(* CODESYS project 1002_xlh_stamp_button_switch_led_manager.project
   Description: Receives some incoming messages and echoes them with CAN-ID +1
   Company: 3S - Smart Software Solutions GmbH
   Version: 1.0.0.0
   Title: CAN Bus API Example
   Author: 3S - Smart Software Solutions GmbH

Project tree, tasks and I/O mapping:
  xLH_base : CODESYS Control for Raspberry Pi 64 SL, CODESYS, order no. 2302000009, version 4.18.0.0
    application app
      libraries: Standard, 3.5.18.0 (System); Util, 3.5.21.0 (System); VisuDialogs, * (System); Memory, * (3S - Smart Software Solutions GmbH); CmpBitmapPool, * (System); CAN API, 1.0.0.4 (CODESYS); MemoryUtils, * (3S - Smart Software Solutions GmbH); CAA CiA 405, 4.3.0.0 (CODESYS)
      task MAIN_TASK (cyclic, interval 10 ms, priority 1) calls ExpeditedReadExample, MAIN
      program MAIN [ST]
      trace Trace_Switch (task MAIN_TASK): MAIN.byDigOutButton, MAIN.byDigInButton, MAIN.fbReadStatusLoopTime.diValue
      function block FB_SDO_READ_4_BYTE [ST]
      CO_API/
        program ExpeditedReadExample [ST]
        program ExpeditedWriteExample [ST]
    SoftMotion General Axis Pool
      a_axis : SM_Drive_PosControl, CODESYS, order no. 1805, version 4.18.0.0
          settings: wDriveID = 4; dwRatioTechUnitsDenom = 101846; iRatioTechUnitsNum = -125; eRampType = 1; fSWMaxVelocity = 50; fSWMaxAcceleration = 100; fSWMaxDeceleration = 100; fSWMaxJerk = 1000; fSWLimitNegative = -1000.0; ScalingIncs = 814768; ScalingUnits = 1000; InvertDirection = TRUE; IsLinearMotor = TRUE; MaximumOutputVelocityInt = 40738; MinimumOutputVelocityInt = -40738; Kp = 0.05; MaxFollowingError = 5.0; EnableFollowingErrorCheck = TRUE; DeadTime = 3.0
      x_axis : SM_Drive_PosControl, CODESYS, order no. 1805, version 4.18.0.0
          settings: dwRatioTechUnitsDenom = 101846; iRatioTechUnitsNum = 125; eRampType = 1; fSWMaxVelocity = 50; fSWMaxAcceleration = 100; fSWMaxDeceleration = 100; fSWMaxJerk = 1000; fSWLimitNegative = -1000; ScalingIncs = 814768; ScalingUnits = 1000; IsLinearMotor = TRUE; MaximumOutputVelocityInt = 40738; MinimumOutputVelocityInt = -40738; Kp = 0.05; MaxFollowingError = 5.0; EnableFollowingErrorCheck = TRUE; DeadTime = 3.0
      y_axis : SM_Drive_PosControl, CODESYS, order no. 1805, version 4.18.0.0
          settings: wDriveID = 2; dwRatioTechUnitsDenom = 101846; iRatioTechUnitsNum = 125; eRampType = 1; fSWMaxVelocity = 50; fSWMaxAcceleration = 100; fSWMaxDeceleration = 100; fSWMaxJerk = 1000; fSWLimitNegative = -1000; ScalingIncs = 814768; ScalingUnits = 1000; IsLinearMotor = TRUE; MaximumOutputVelocityInt = 40738; MinimumOutputVelocityInt = -40738; Kp = 0.05; MaxFollowingError = 5.0; EnableFollowingErrorCheck = TRUE; DeadTime = 3.0
      z_axis : SM_Drive_PosControl, CODESYS, order no. 1805, version 4.18.0.0
          settings: wDriveID = 3; dwRatioTechUnitsDenom = 101846; iRatioTechUnitsNum = 125; eRampType = 1; fSWMaxVelocity = 50; fSWMaxAcceleration = 100; fSWMaxDeceleration = 100; fSWMaxJerk = 1000; fSWLimitNegative = -1000; ScalingIncs = 814768; ScalingUnits = 1000; IsLinearMotor = TRUE; MaximumOutputVelocityInt = 40738; MinimumOutputVelocityInt = -40738; Kp = 0.05; MaxFollowingError = 5.0; EnableFollowingErrorCheck = TRUE; DeadTime = 3.0
    GPIOs_A_B : GPIOs B+/Pi2, CODESYS, version 4.18.0.0
        unmapped channels: digital inputs (GPIO0..GPIO31), digital outputs (GPIO0..GPIO31)
    Onewire
    Camera device
      <Leer>
    SPI
    I²C
    CANbus : CANbus, CODESYS, version 4.3.0.0
        settings: Baudrate = 1000 kbit/s
      CANopen_Manager : CANopen_Manager, CODESYS, version 4.3.0.0
          settings: ConfigVersion = 50659584
        xlh_digital_switch_button_led : xlh_digital_switch_button_led, xemax ag, order no. 0, version Revision=16#00000001, FileVersion=1.0
            settings: NODEIDSAVED = 1; SDO Timeout = 1000000; PDO_Autoconfig = FALSE; EXPERTSETTINGS = False; Sync-General Parameters.Sync-COBID = 16#00000080; Sync-General Parameters.Communication Cycle Period = 16#00000000 usec; PDO 16#1400.COBID = 16#00000201; Process by CANopenManager = TRUE; PDO 16#1800.COBID = 16#00000181; Process by CANopenManager = TRUE; Leds Button.Subindex = 16#01; Leds Switch.Subindex = 16#01; Digital Inputs Button.Subindex = 16#01; Digital Inputs Switch.Subindex = 16#01; SDO List.Set COB-ID sync.Index = 16#1005; SDO List.Set COB-ID sync.Subindex = 16#00; SDO List.Set COB-ID sync.Value = 16#00000080; SDO List.Set COB-ID sync.Size = 32; SDO List.Set COB-ID sync.AbortIfError = FALSE; SDO List.Set COB-ID sync.JumpToLine = FALSE; SDO List.Set COB-ID sync.Line = 0; SDO List.Set communication cycle period.Index = 16#1006; SDO List.Set communication cycle period.Subindex = 16#00; SDO List.Set communication cycle period.Value = 16#00000000; SDO List.Set communication cycle period.Size = 32; SDO List.Set communication cycle period.AbortIfError = FALSE; SDO List.Set communication cycle period.JumpToLine = FALSE; SDO List.Set communication cycle period.Line = 0; SDO List.Set Guardtime.Index = 16#100C; SDO List.Set Guardtime.Subindex = 16#00; SDO List.Set Guardtime.Value = 16#000000C8; SDO List.Set Guardtime.Size = 16; SDO List.Set Guardtime.AbortIfError = FALSE; SDO List.Set Guardtime.JumpToLine = FALSE; SDO List.Set Guardtime.Line = 0; SDO List.Set Lifetime.Index = 16#100D; SDO List.Set Lifetime.Subindex = 16#00; SDO List.Set Lifetime.Value = 16#00000003; SDO List.Set Lifetime.Size = 8; SDO List.Set Lifetime.AbortIfError = FALSE;
              SDO List.Set Lifetime.JumpToLine = FALSE; SDO List.Set Lifetime.Line = 0; SDO List.Set Heartbeat Consumer.Index = 16#1016; SDO List.Set Heartbeat Consumer.Subindex = 16#01; SDO List.Set Heartbeat Consumer.Value = 0; SDO List.Set Heartbeat Consumer.Size = 32; SDO List.Set Heartbeat Consumer.AbortIfError = FALSE; SDO List.Set Heartbeat Consumer.JumpToLine = FALSE; SDO List.Set Heartbeat Consumer.Line = 0; SDO List.Disable PDO.Index = 16#1400; SDO List.Disable PDO.Subindex = 16#01; SDO List.Disable PDO.Value = 16#80000201; SDO List.Disable PDO.Size = 32; SDO List.Disable PDO.AbortIfError = FALSE; SDO List.Disable PDO.JumpToLine = FALSE; SDO List.Disable PDO.Line = 0; SDO List.Set transmission type.Index = 16#1400; SDO List.Set transmission type.Subindex = 16#02; SDO List.Set transmission type.Value = 16#FF; SDO List.Set transmission type.Size = 8; SDO List.Set transmission type.AbortIfError = FALSE; SDO List.Set transmission type.JumpToLine = FALSE; SDO List.Set transmission type.Line = 0; SDO List.Set and enable COB-ID.Index = 16#1400; SDO List.Set and enable COB-ID.Subindex = 16#01; SDO List.Set and enable COB-ID.Value = 16#00000201; SDO List.Set and enable COB-ID.Size = 32; SDO List.Set and enable COB-ID.AbortIfError = FALSE; SDO List.Set and enable COB-ID.JumpToLine = FALSE; SDO List.Set and enable COB-ID.Line = 0; SDO List.Disable PDO.Index = 16#1800; SDO List.Disable PDO.Subindex = 16#01; SDO List.Disable PDO.Value = 16#80000181; SDO List.Disable PDO.Size = 32; SDO List.Disable PDO.AbortIfError = FALSE; SDO List.Disable PDO.JumpToLine = FALSE; SDO List.Disable PDO.Line = 0; SDO List.Set transmission type.Index = 16#1800; SDO List.Set transmission type.Subindex = 16#02; SDO List.Set transmission type.Value = 16#FF;
              SDO List.Set transmission type.Size = 8; SDO List.Set transmission type.AbortIfError = FALSE; SDO List.Set transmission type.JumpToLine = FALSE; SDO List.Set transmission type.Line = 0; SDO List.Set inhibit time.Index = 16#1800; SDO List.Set inhibit time.Subindex = 16#03; SDO List.Set inhibit time.Value = 16#0000; SDO List.Set inhibit time.Size = 16; SDO List.Set inhibit time.AbortIfError = FALSE; SDO List.Set inhibit time.JumpToLine = FALSE; SDO List.Set inhibit time.Line = 0; SDO List.Set event time.Index = 16#1800; SDO List.Set event time.Subindex = 16#05; SDO List.Set event time.Value = 16#0000; SDO List.Set event time.Size = 16; SDO List.Set event time.AbortIfError = FALSE; SDO List.Set event time.JumpToLine = FALSE; SDO List.Set event time.Line = 0; SDO List.Set and enable COB-ID.Index = 16#1800; SDO List.Set and enable COB-ID.Subindex = 16#01; SDO List.Set and enable COB-ID.Value = 16#00000181; SDO List.Set and enable COB-ID.Size = 32; SDO List.Set and enable COB-ID.AbortIfError = FALSE; SDO List.Set and enable COB-ID.JumpToLine = FALSE; SDO List.Set and enable COB-ID.Line = 0; ConfigVersion = 50659584
            output app.MAIN.byDigOutButton : USINT  // Digital Outputs Button
            output app.MAIN.byDigOutSwitch : USINT  // Digital Outputs Switch
            input  app.MAIN.byDigInButton : USINT  // Digital Inputs Button
            input  app.MAIN.byDigInSwitch : USINT  // Digital Inputs Switch
  libraries: VisuSymbols, 4.5.0.0 (System); DepictorBase, 1.2.0.0 (CODESYS)
  text list GlobalTextList
  5ce3da45-db07-42e7-a21c-a00fff4ed8f6|C:\Users\phe\Downloads\Musterloesung_FUP.PNG
*)

// xLH_base/app/CO_API/ExpeditedReadExample
// The following program reads the device type of CANopenRemoteDevice and shows how to usde SDORead4 function block.
// Set xEnable to TRUE in online mode to get the program working.
PROGRAM ExpeditedReadExample
VAR
	xEnable       : BOOL; // Set this variable to true to start the example code. Variable will be set to FALSE if Expedited transfer finished execution.
	dwValue : DWORD; //read value
	dwAbortCode : DWORD; //contains abort code in case of error
	
	SDORead4 	  : CIA405.SDO_READ4;
END_VAR

IF SDORead4.CONFIRM THEN
	//value was read without error
	// ==> Copy data from SDO read function block
	MEMUtils.MemCpy(pbyDest := ADR(dwValue), pbySrc := ADR(SDORead4.DATA[1]), dwSize := SIZEOF(dwValue));
	//==> On big endian systems: dwValue has to be swapped to CANopen byte order (= Little Endian).
	//MEMUtils.SwapLocalToIntel(pAddress := ADR(dwValue), iSize := TO_INT(SIZEOF(dwValue))); //function only swaps on big endian systems
	xEnable := FALSE;
ELSIF SDORead4.ERROR <> CiA405.CANOPEN_KERNEL_ERROR.CANOPEN_KERNEL_NO_ERROR THEN
	//Error occured
	IF SDORead4.ERROR = CIA405.CANOPEN_KERNEL_ERROR.CANOPEN_KERNEL_OTHER_ERROR THEN
		//output error info contains abort code in little endian format
		MEMUtils.MemCpy(pbyDest := ADR(dwAbortCode), pbySrc := ADR(SDORead4.ERRORINFO), dwSize := SIZEOF(dwAbortCode));
		MEMUtils.SwapLocalToIntel(pAddress := ADR(dwAbortCode), iSize := TO_INT(SIZEOF(dwAbortCode))); //function only swaps on big endian systems	
	END_IF
	xEnable := FALSE;
END_IF

SDORead4(
	NETWORK:= CANbus.NetId + 1, //CODESYS NetId starts by 0 (the number entered into the CANbus configurator); CiA405 NETWORK by 1; That is the reason why we have to increment it here.
	ENABLE:= xEnable,
	TIMEOUT:= 0, //Timeout for SDO read in ms. Here: 0 ==> no timeout
	DEVICE:= xLH_digital_switch_button_led.NodeID, // NodeID of destination device
	CHANNEL:= 0, //SDO channel which should be used. 0 means auto channeling ==> the next free channel will be used. It depends on the slave which settings are working here but 0 and channel 1 is always working. 
	INDEX:= 16#5800, //object index which should be read
	SUBINDEX:= 2 //object sub index which should be read
);

END_PROGRAM

// xLH_base/app/MAIN
PROGRAM MAIN
VAR
	byDigInSwitch: USINT;
	byDigOutSwitch: USINT;
	byDigInButton: USINT;
	byDigOutButton: USINT;
	byDummy: USINT;
	udiDummy: UDINT;
	
	fbBlink: BLINK := (TIMEHIGH:=T#100MS, TIMELOW:=T#100MS, ENABLE:=TRUE);
	fbReadStatusRefreshTime: FB_SDO_READ_4_BYTE;
	fbReadStatusLoopTime: FB_SDO_READ_4_BYTE;
END_VAR

byDummy := byDigInButton;
byDigOutButton := byDigOutButton + 1;

byDummy := byDigInSwitch;
byDigOutSwitch := byDigInSwitch OR byDigInButton;

fbBlink();
fbReadStatusRefreshTime(
	bEnable:=fbBlink.OUT,
	usCoDeviceId:=xlh_digital_switch_button_led.NodeID,
	uiIndex:=16#5800, usSubindex:=1);
fbReadStatusLoopTime(
	bEnable:= NOT fbBlink.OUT,
	usCoDeviceId:=xlh_digital_switch_button_led.NodeID,
	uiIndex:=16#5800, usSubindex:=2);
udiDummy := fbReadStatusRefreshTime.udiValue;
udiDummy := fbReadStatusLoopTime.udiValue;

END_PROGRAM

// xLH_base/app/FB_SDO_READ_4_BYTE
FUNCTION_BLOCK FB_SDO_READ_4_BYTE
VAR_INPUT
	bEnable: BOOL;
	usCoDeviceId: USINT;
	usNetId: USINT := 0;
	uiIndex: UINT;
	usSubindex: USINT;
END_VAR
VAR_OUTPUT
	bDone: BOOL;
	bError: BOOL;
	diValue: DINT;
	udiValue: UDINT;
END_VAR
VAR
	dwAbortCode : DWORD; //contains abort code in case of error
	fbSdoRead4Byte: CIA405.SDO_READ4;	
	fbRtEnable: R_TRIG;
END_VAR

fbRtEnable(CLK:=bEnable);
IF fbRtEnable.CLK THEN
	//bEnable := FALSE;
	bDone := FALSE;
	bError := FALSE;
END_IF

IF fbSdoRead4Byte.CONFIRM THEN
	//value was read without error
	// ==> Copy data from SDO read function block
	MEMUtils.MemCpy(pbyDest := ADR(diValue), pbySrc := ADR(fbSdoRead4Byte.DATA[1]), dwSize := SIZEOF(diValue));
	MEMUtils.MemCpy(pbyDest := ADR(udiValue), pbySrc := ADR(fbSdoRead4Byte.DATA[1]), dwSize := SIZEOF(udiValue));
	//==> On big endian systems: dwValue has to be swapped to CANopen byte order (= Little Endian).
	//MEMUtils.SwapLocalToIntel(pAddress := ADR(diValue), iSize := TO_INT(SIZEOF(diValue))); //function only swaps on big endian systems
	//MEMUtils.SwapLocalToIntel(pAddress := ADR(udiValue), iSize := TO_INT(SIZEOF(udiValue))); //function only swaps on big endian systems
	bDone := TRUE;
	bError := FALSE;
ELSIF fbSdoRead4Byte.ERROR <> CiA405.CANOPEN_KERNEL_ERROR.CANOPEN_KERNEL_NO_ERROR THEN
	//Error occured
	IF fbSdoRead4Byte.ERROR = CIA405.CANOPEN_KERNEL_ERROR.CANOPEN_KERNEL_OTHER_ERROR THEN
		//output error info contains abort code in little endian format
		MEMUtils.MemCpy(pbyDest := ADR(dwAbortCode), pbySrc := ADR(fbSdoRead4Byte.ERRORINFO), dwSize := SIZEOF(dwAbortCode));
		MEMUtils.SwapLocalToIntel(pAddress := ADR(dwAbortCode), iSize := TO_INT(SIZEOF(dwAbortCode))); //function only swaps on big endian systems	
	END_IF
	bDone := FALSE;
	bError := TRUE;
END_IF

fbSdoRead4Byte(
	NETWORK:= CANbus.NetId + 1, //CODESYS NetId starts by 0 (the number entered into the CANbus configurator); CiA405 NETWORK by 1; That is the reason why we have to increment it here.
	ENABLE:= fbRtEnable.CLK,
	TIMEOUT:= 0, //Timeout for SDO read in ms. Here: 0 ==> no timeout
	DEVICE:= usCoDeviceId, // NodeID of destination device
	CHANNEL:= 0, //SDO channel which should be used. 0 means auto channeling ==> the next free channel will be used. It depends on the slave which settings are working here but 0 and channel 1 is always working. 
	INDEX:= uiIndex, //object index which should be read
	SUBINDEX:= usSubindex //object sub index which should be read
);

END_FUNCTION_BLOCK

// xLH_base/app/CO_API/ExpeditedWriteExample
// The following program writes a 32bit value with SDO expedited transfer.
// Set xEnable to TRUE in online mode to get the program working.
PROGRAM ExpeditedWriteExample
VAR
	xEnable       : BOOL; // Set this variable to true to start the example code. Variable will be set to FALSE if Expedited transfer finished execution.
	diValue : DINT := 10; //value which should be written
	dwAbortCode : DWORD; //contains abort code in case of error
	
	SDOWrite4 	  : CiA405.SDO_WRITE4;
	RTrig 		  : Standard.R_TRIG;
END_VAR

RTrig(CLK := xEnable); //detect a rising edge for xEnable

IF RTrig.Q THEN
	// Rising edge for xEnable detected ==> Prepare SDO write function block
	// ==> Copy data to SDO write function block
	MEMUtils.MemCpy(pbyDest := ADR(SDOWrite4.DATA[1]), pbySrc := ADR(diValue), dwSize := SIZEOF(diValue));
	//==> On big endian systems: diValue has to be swapped to CANopen byte order (= Little Endian).
	MEMUtils.SwapLocalToIntel(pAddress := ADR(SDOWrite4.DATA[1]), iSize := TO_INT(SIZEOF(diValue))); //function only swaps on big endian systems
END_IF

IF SDOWrite4.CONFIRM THEN
	//value was written without error
	xEnable := FALSE;
ELSIF SDOWrite4.ERROR <> CiA405.CANOPEN_KERNEL_ERROR.CANOPEN_KERNEL_NO_ERROR THEN
	//Error occured
	IF SDOWrite4.ERROR = CIA405.CANOPEN_KERNEL_ERROR.CANOPEN_KERNEL_OTHER_ERROR THEN
		//output error info contains abort code in little endian format
		MEMUtils.MemCpy(pbyDest := ADR(dwAbortCode), pbySrc := ADR(SDOWrite4.ERRORINFO), dwSize := SIZEOF(dwAbortCode));
		MEMUtils.SwapLocalToIntel(pAddress := ADR(dwAbortCode), iSize := TO_INT(SIZEOF(dwAbortCode))); //function only swaps on big endian systems	
	END_IF
	xEnable := FALSE;
END_IF

SDOWrite4(
	NETWORK:= CANbus.NetId + 1, //CODESYS NetId starts by 0 (the number entered into the CANbus configurator); CiA405 NETWORK by 1; That is the reason why we have to increment it here.
	ENABLE:= xEnable,
	TIMEOUT:= 0, //Timeout for SDO write in ms. Here: 0 ==> no timeout
	DEVICE:= xLH_digital_switch_button_led.NodeID, // NodeID of destination device
	CHANNEL:= 0, //SDO channel which should be used. 0 means auto channeling ==> the next free channel will be used. It depends on the slave which settings are working here but 0 and channel 1 is always working. 
	INDEX:= 16#6412, //object index which should be written
	SUBINDEX:= 1, //object sub index which should be written
	DATALENGTH:= TO_USINT(SIZEOF(diValue)) //length of data to be written
);

END_PROGRAM
